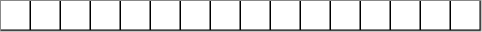
VISUALIZATION WordBitDisplay  // 482x32
VAR_IN_OUT
	nVal	:	WORD;
END_VAR
    Rectangle (0,0 30x30), colour toggle: nVal.15
    Rectangle (30,0 30x30), colour toggle: nVal.14
    Rectangle (60,0 30x30), colour toggle: nVal.13
    Rectangle (90,0 30x30), colour toggle: nVal.12
    Rectangle (120,0 30x30), colour toggle: nVal.11
    Rectangle (150,0 30x30), colour toggle: nVal.10
    Rectangle (180,0 30x30), colour toggle: nVal.9
    Rectangle (210,0 30x30), colour toggle: nVal.8
    Rectangle (240,0 30x30), colour toggle: nVal.7
    Rectangle (270,0 30x30), colour toggle: nVal.6
    Rectangle (300,0 30x30), colour toggle: nVal.5
    Rectangle (330,0 30x30), colour toggle: nVal.4
    Rectangle (360,0 30x30), colour toggle: nVal.3
    Rectangle (390,0 30x30), colour toggle: nVal.2
    Rectangle (420,0 30x30), colour toggle: nVal.1
    Rectangle (450,0 30x30), colour toggle: nVal.0
END_VISUALIZATION

(* stored: Version 1.1.0.1, ProductVersion 3.1.4024.0
   Visu WordBitDisplay: Id {d6d3276f-24d6-0a97-2d85-81b9e893839f} *)
